(* IEC 61131-3 sources: BODAS-HelloWorld/extracted_st/bodas_rc18_12_40/plc_logic/application/02_easyconfig/easyconfig_import/bds_out_ec/bds_out_ec_gvl, 1 file *)

(* ---- bds_out_ec_gvl.st ---- *)
(* --- Interface --- *)
{attribute 'qualified_only' := ''}
VAR_GLOBAL CONSTANT
    RECONF_X_X_X25 : UDINT := 0;
END_VAR
